RoboDK station: multipasswelding_RBT23IT057.rdk

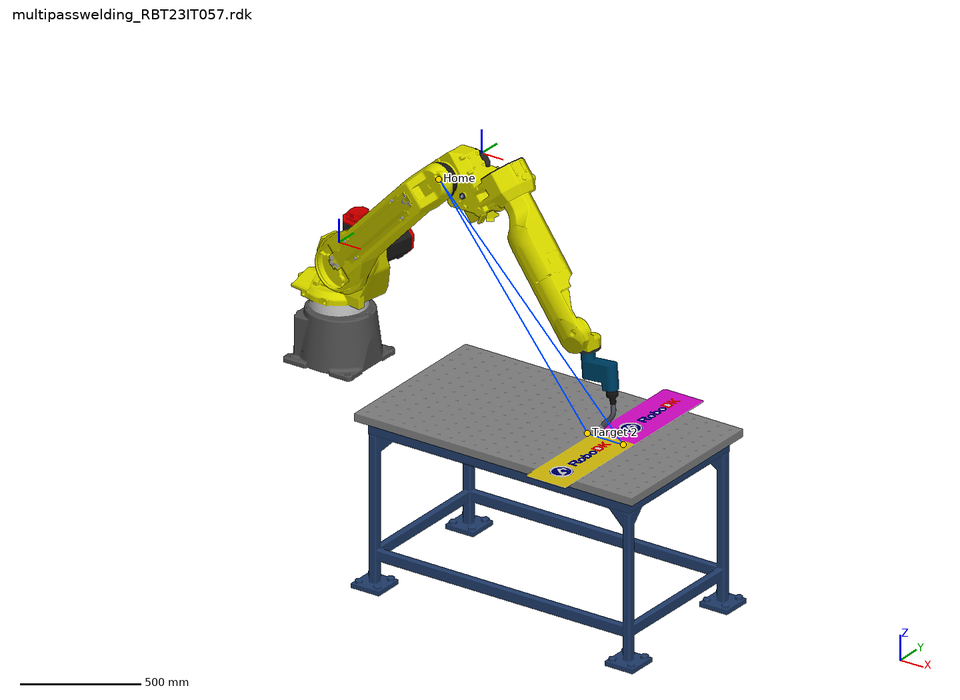
[picture v0: the station drawn from its stored meshes, robots at their saved joint values, targets as dots, program paths as lines]
Station multipasswelding_RBT23IT057 (saved by RoboDK 5.9.2). Poses are relative to the parent item; angles as X-Y-Z fixed-axis rotations.
  - frame Fanuc ARC Mate 120iC Base at (0, 0, 0) mm
    - target Home (joint target) at (503.79, 0, 431.51) mm, rotated rx -180 ry -40.14 rz 180 deg; joints [0, -40.164, 3.259, 0, -88.402, 180] of Fanuc ARC Mate 120iC
    - robot Fanuc ARC Mate 120iC: 6 axes, payload 3 kg, reach 1811 mm, repeatability 0.08 mm, weight 250 kg
        modified DH rows (alpha deg, a mm, theta deg, d mm): 0, 0, 0, 525; -90, 150, -90, 0; 0, 790, 0, 0; -90, 250, 0, 835; 90, 0, 0, 0; -90, 0, 0, 100
        base shift (0, 0, -525) mm
        joint limits [-185, -100, -345, -200, -140, -450] to [185, 160, 375.6, 200, 140, 450]; home [0, 0, 0, 0, 0, 0]; saved at [-9.675, 44.385, -49.273, -1.389, -35.947, 190.766]
      - tool Weld gun, TCP at (26, -10, 371.3) mm, rotated rx 20 ry 75 rz 0 deg, size 299.9 x 60 x 318.3 mm
    - target Target 2 (Cartesian target) at (1430.4, -251.48, -376.91) mm, rotated rx -160 ry -70.14 rz -180 deg; joints [-9.675, 44.385, -49.273, -1.389, -35.947, 190.766] of Fanuc ARC Mate 120iC
    - target Target 3 (Cartesian target) at (1611.44, -251.48, -378.15) mm, rotated rx -160 ry -70.14 rz -180 deg; joints [-8.596, 56.922, -39.449, -1.012, -45.753, 189.272] of Fanuc ARC Mate 120iC
  - object Table 1400x800x800mm at (880, -260, -370) mm, size 1420 x 820 x 800 mm, geometry from Table-1400x800x800mm.sld
  - frame Frame 2 at (0, 1030, 0) mm
    - object RoboDK Nametag Plate 500x200mm at (1660, -1770, -370) mm, size 200 x 500 x 5 mm, geometry from RoboDK-Nametag-Plate-500x200mm.sld
    - object RoboDK Nametag Plate 500x200mm at (1660, -1270, -370) mm, size 200 x 500 x 5 mm, geometry from RoboDK-Nametag-Plate-500x200mm.sld
  - program Prog1 (15 instructions, listed below)
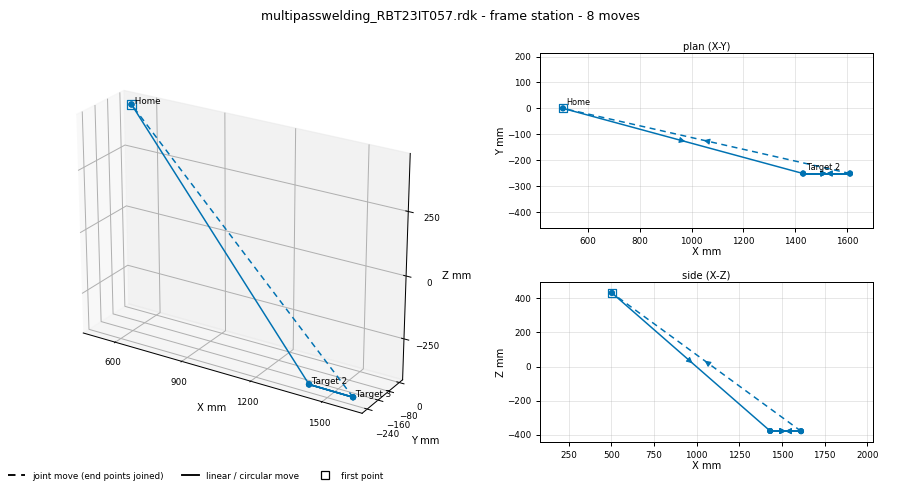
[picture p0: tool path of multipasswelding_RBT23IT057.rdk in frame station, 8 of 8 moves have a stored position in this frame; points joined in program order, loops and branches not executed]

--- program Prog1 (robot Fanuc ARC Mate 120iC) ---
  Set Ref.: Fanuc ARC Mate 120iC Base
  Set Tool: Weld gun
  MoveJ (Home)
  MoveL (Target 2)
  MoveL (Target 3)
  Pause 500 ms
  MoveL (Target 2)
  Pause 500 ms
  MoveL (Target 3)
  Pause 500 ms
  MoveL (Target 2)
  Pause 500 ms
  MoveL (Target 3)
  Pause 500 ms
  MoveJ (Home)
